// TIA Portal project "Herz_3_pontos" (V13)

(* hardware
DEVICE "S7300/ET200M station_1"  S7-300 station
   slot 0: "Rail_0"  Rail  6ES7 390-1***0-0AA0
   slot 1: "PS 307 5A_1"  PS 307 5A  6ES7 307-1EA01-0AA0
   slot 2: "PLC_1"  CPU 314C-2 PN/DP  6ES7 314-6EH04-0AB0  V3.3
      slot 2: "PROFINET interface_1"  PN-IO
         slot 1: "Port_1"  Port
         slot 2: "Port_2"  Port
      slot 5: "DI 24/DO 16_1"  DI24/DO16
      slot 6: "AI 5/AO 2_1"  AI5/AO2
      slot 7: "Count_1"  Counter
      slot 8: "Positioning_1"  Positioning
*)

// ===== PLC "PLC_1"  CPU 314C-2 PN/DP =====

VAR_GLOBAL   // PLC tag table "Default tag table"
   "sr1" AT %I0.0 : Bool;
   "sr2" AT %I0.1 : Bool;
   "sr3" AT %I0.2 : Bool;
   "esteira1" AT %Q0.0 : Bool;
   "esteira2" AT %Q0.1 : Bool;
END_VAR

ORGANIZATION_BLOCK "Main"   // OB1, LAD
TITLE = "Main Program Sweep (Cycle)"
{ S7_Optimized_Access := 'FALSE' }
VERSION : 0.1
   VAR_TEMP
      OB1_EV_CLASS : Byte;   // Bits 0-3 = 1 (Coming event), Bits 4-7 = 1 (Event class 1)
      OB1_SCAN_1 : Byte;   // 1 (Cold restart scan 1 of OB 1), 3 (Scan 2-n of OB 1)
      OB1_PRIORITY : Byte;   // Priority of OB Execution
      OB1_OB_NUMBR : Byte;   // 1 (Organization block 1, OB1)
      OB1_RESERVED_1 : Byte;   // Reserved for system
      OB1_RESERVED_2 : Byte;   // Reserved for system
      OB1_PREV_CYCLE : Int;   // Cycle time of previous OB1 scan (milliseconds)
      OB1_MIN_CYCLE : Int;   // Minimum cycle time of OB1 (milliseconds)
      OB1_MAX_CYCLE : Int;   // Maximum cycle time of OB1 (milliseconds)
      OB1_DATE_TIME : Date_And_Time;   // Date and time OB1 started
   END_VAR
BEGIN

REGION Network 1
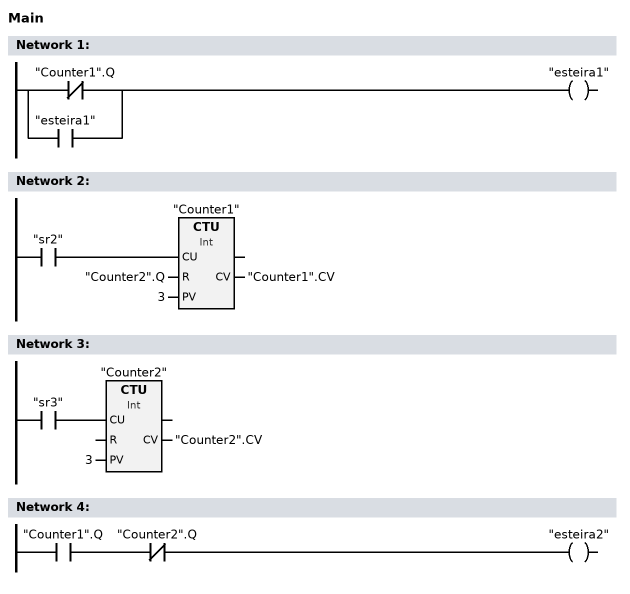
   RUNG wire#powerrail
      I_Contact( "Counter1".Q )
      wire#w1
      Coil( "esteira1" )
   END_RUNG
   RUNG wire#powerrail
      Contact( "esteira1" )
   END_RUNG wire#w1
   // the same network as SCL:
   "esteira1" := NOT "Counter1".Q OR "esteira1";
END_REGION

REGION Network 2
   "Counter1".CTU(CU := "sr2", R := "Counter2".Q, PV := 3, CV => "Counter1".CV);
END_REGION

REGION Network 3
   "Counter2".CTU(CU := "sr3", PV := 3, CV => "Counter2".CV);
END_REGION

REGION Network 4
   RUNG wire#powerrail
      Contact( "Counter1".Q )
      I_Contact( "Counter2".Q )
      Coil( "esteira2" )
   END_RUNG
   // the same network as SCL:
   "esteira2" := "Counter1".Q AND NOT "Counter2".Q;
END_REGION
END_ORGANIZATION_BLOCK